// TIA Portal V16 export
// export: Created 2024-05-10T06:46:43.4529038Z, ExportSetting WithDefaults, DisplayName Totally Integrated Automation Portal, DisplayVersion V16, DisplayName TIA Portal Version Control Interface, DisplayVersion V16, DisplayName TIA Portal Openness, DisplayVersion V16, DisplayName STEP 7 Professional, DisplayVersion V16, DisplayName STEP 7 Safety, DisplayVersion V16, DisplayName WinCC Professional, DisplayVersion V16
DATA_BLOCK "K07_轴组_DB"   // DB7
VERSION : 0.1
// stored: AutoNumber true, DBAccessibleFromOPCUA true, InstanceOfName K07_轴组, InstanceOfType FB
"K07_轴组"
   // VAR
   //    Axis1Write { S7_SetPoint := 'True'} : "F121_SinaParaWrite(SV660F)";
   //    Axis1Pos { S7_SetPoint := 'True'} : "F120_SinaPos(SV660F)";
   // END_VAR
BEGIN
END_DATA_BLOCK
